// TIA Portal V19 export
DATA_BLOCK "LEVEL_TRANSMITTER-801"   // DB14
// stored: InstanceOfName SCALE, InstanceOfType FB
"SCALE"
   // VAR_INPUT
   //    "SCALE MIN" : Real;
   //    "SCALE MAX" : Real;
   //    INPUT : Int;
   //    "RAW MIN" : Int;
   //    "RAW MAX" : Int;
   // END_VAR
   // VAR_OUTPUT
   //    "PV VALUE" : Real;
   // END_VAR
BEGIN
END_DATA_BLOCK
